PROGRAM PRG_TEST
VAR
	fbEventBuffer_Test : FB_EventBuffer_Test;
END_VAR

TcUnit.RUN();

END_PROGRAM

(* stored: Version 1.1.0.1, ProductVersion 3.1.4024.12
   POU PRG_TEST: Id {137101cf-2f09-4096-8f05-41d2c6fe9e05}, SpecialFunc None *)
